(* PLC project ifmCR711S_TemplateProject, CODESYS CODESYS V3.5 SP11 Patch 5 *)
(* stored: creationDateTime 2026-05-10T19:29:40.3172001, version 2.4.10.0, modificationDateTime 2026-05-10T19:24:10.3108894, organization ifm electronic *)
(* Project template with CR711S configured 2.25MByte Standard 2.25MByte Safety *)

(* values of EControlMode: INIT: Initial state when starting ferry *)

{attribute 'qualified_only'}
{attribute 'strict'}
TYPE EControlMode : (INIT, MANUAL, REMOTE, AUTO, REMOTE_MOBILE, FAILSAFE);
END_TYPE

(* values of ETransitionState: STABLE: No switch in progress *)

(* Where the system is in the switch process *)
{attribute 'qualified_only'}
{attribute 'strict'}
TYPE ETransitionState : (INIT, STABLE, PRE_TAKEOVER, VALIDATE_TAKEOVER, FAILSAFE);
END_TYPE

(* values of EPendingMode: NONE: No state pending; PENDING_MANUAL: Pending manual; PENDING_REMOTE: Pending remote; PENDING_AUTO: Pending auto *)

{attribute 'qualified_only'}
{attribute 'strict'}
TYPE EPendingMode : (NONE, PENDING_MANUAL, PENDING_REMOTE, PENDING_AUTO, PENDING_REMOTE_MOBILE);
END_TYPE

PROGRAM PLC_PRG
  VAR
    fbMonitoringChannel : MonitoringChannel;
    fbShutdownService : ShutdownService;
  END_VAR

                    fbMonitoringChannel(
	HB_Manual_OK := EVL.HB_Manual_OK, 
	HB_Remote_OK := EVL.HB_Remote_OK,
	HB_Auto_OK	 := EVL.HB_Auto_OK, 
	HB_Remote_Mobile_OK := EVL.HB_Remote_Mobile_OK
);

fbShutdownService( 
	EmergencyShutdown := fbMonitoringChannel.EmergencyShutdown
); 
                  
END_PROGRAM

FUNCTION_BLOCK MonitoringChannel
  VAR_INPUT
    HB_Manual_OK : BOOL;
    HB_Remote_OK : BOOL;
    HB_Auto_OK : BOOL;
    HB_Remote_Mobile_OK : BOOL;
  END_VAR
  VAR_OUTPUT
    EmergencyShutdown : BOOL;
  END_VAR
  VAR
    HB_Manual_Fail : BOOL;
    HB_Remote_Fail : BOOL;
    HB_Auto_Fail : BOOL;
    HB_Remote_Mobile_Fail : BOOL;
  END_VAR

                    
HB_Manual_Fail := NOT HB_Manual_OK; 
HB_Remote_Fail := NOT HB_Remote_OK; 
HB_Auto_Fail   := NOT HB_Auto_OK;
HB_Remote_Mobile_Fail := NOT HB_Remote_Mobile_OK; 

IF HB_Manual_Fail AND HB_Remote_Fail AND HB_Auto_Fail AND HB_Remote_Mobile_Fail THEN 
	EmergencyShutdown := TRUE; 
END_IF


                  
END_FUNCTION_BLOCK

FUNCTION_BLOCK ShutdownService
  VAR_INPUT
    EmergencyShutdown : BOOL;
  END_VAR
  VAR
    Alert : BOOL;
  END_VAR

                    //Once triggered, the alert stays TRUE until system restart

IF EmergencyShutdown THEN 
	Alert := TRUE; 
END_IF
                  
END_FUNCTION_BLOCK

PROGRAM PLC_PRG
  VAR
    fbInputProcessing : InputProcessing;
    fbControlUnit : ControlUnit;
    fbOutputProcessing : OutputProcessing;
    fbIntegrityCheck : IntegrityCheck;
    fbDecisionLogger : DecisionLogger;
    fbHBGen_Manual : FB_HeartBeatGenerator;
    fbHBGen_Remote : FB_HeartBeatGenerator;
    fbHBGen_Auto : FB_HeartBeatGenerator;
    fbHBGen_Remote_Mobile : FB_HeartBeatGenerator;
    fbHB_Manual : FB_HeartBeat;
    fbHB_Remote : FB_HeartBeat;
    fbHB_Auto : FB_HeartBeat;
    fbHB_Remote_Mobile : FB_HeartBeat;
  END_VAR

                    CR710S_Config(); 			//IO Configuration

IOWrapper.READ_INPUTS(); 	//Call IOWrapper Main Program and Read Data from Inputs   

fbInputProcessing(
	xReqManual 			:= GVL_IO.ReqManual,
	xAckManual 			:= GVL_IO.AckManual, 
	xRelManual 			:= GVL_IO.RelManual, 
	xHB_Manual			:= IN0103.VAR_OUT.xValueDigital, 
	xReqRemote			:= GVL_IO.ReqRemote, 
	xAckRemote			:= GVL_IO.AckRemote, 
	xRelRemote        	:= GVL_IO.RelRemote,
	xHB_Remote        := GVL_HeartBeat.HB_Remote_Signal,
	xReqAuto          := GVL_IO.ReqAuto,
    xAckAuto          := GVL_IO.AckAuto,
    xRelAuto          := GVL_IO.RelAuto,
    xHB_Auto          := GVL_HeartBeat.HB_Auto_Signal,
	xReqRemoteMobile  := GVL_IO.ReqRemoteMobile,
    xAckRemoteMobile  := GVL_IO.AckRemoteMobile,
    xRelRemoteMobile  := GVL_IO.RelRemoteMobile,
    xHB_Remote_Mobile := GVL_HeartBeat.HB_Remote_Mobile_Signal
	
);

fbHB_Manual(xSignal        := fbHBGen_Manual.xSignal);
fbHB_Remote(xSignal        := fbHBGen_Remote.xSignal);
fbHB_Auto(xSignal          := fbHBGen_Auto.xSignal);
fbHB_Remote_Mobile(xSignal := fbHBGen_Remote_Mobile.xSignal);

GVL_HeartBeat.HB_Manual_OK := fbHB_Manual.xOk;
GVL_HeartBeat.HB_Remote_OK := fbHB_Remote.xOk;
GVL_HeartBeat.HB_Auto_OK   := fbHB_Auto.xOk;
GVL_HeartBeat.HB_Remote_Mobile_OK := fbHB_Remote_Mobile.xOk;

//Heartbeat generator
fbHBGen_Manual(); 
fbHBGen_Remote(); 
fbHBGen_Auto();
fbHBGen_Remote_Mobile(); 


fbIntegrityCheck(
    ReqManual        := fbInputProcessing.ReqManual,
    ReqRemote        := fbInputProcessing.ReqRemote,
	ReqAuto			 := fbInputProcessing.ReqAuto,
	ReqRemoteMobile  := fbInputProcessing.ReqRemoteMobile,
    AckManual        := fbInputProcessing.AckManual,
    AckRemote        := fbInputProcessing.AckRemote,
	AckAuto			 := fbInputProcessing.AckAuto,
	AckRemoteMobile  := fbInputProcessing.AckRemoteMobile,
    RelManual        := fbInputProcessing.RelManual,
    RelRemote        := fbInputProcessing.RelRemote,
	RelAuto			 := fbInputProcessing.RelAuto,
	RelRemoteMobile  := fbInputProcessing.RelRemoteMobile,
    HB_Manual_Signal := fbInputProcessing.HB_Manual_Signal,
    HB_Remote_Signal := fbInputProcessing.HB_Remote_Signal,
	HB_Auto_Signal	 := fbInputProcessing.HB_Auto_Signal,
	HB_Remote_Mobile_Signal := fbInputProcessing.HB_Remote_Mobile_Signal, 
);

fbControlUnit(
    ReqManual  		:= fbIntegrityCheck.ReqManual_Out,
	AckManual   	:= fbIntegrityCheck.AckManual_Out,
	RelManual   	:= fbIntegrityCheck.RelManual_Out,
    ReqRemote   	:= fbIntegrityCheck.ReqRemote_Out,
    AckRemote   	:= fbIntegrityCheck.AckRemote_Out,
    RelRemote   	:= fbIntegrityCheck.RelRemote_Out,
	ReqAuto			:= fbIntegrityCheck.ReqAuto_Out,
	AckAuto			:= fbIntegrityCheck.AckAuto_Out,
	RelAuto			:= fbIntegrityCheck.RelAuto_Out,
	ReqRemoteMobile := fbIntegrityCheck.ReqRemoteMobile_Out, 
	AckRemoteMobile := fbIntegrityCheck.AckRemoteMobile_Out, 
	RelRemoteMobile := fbIntegrityCheck.RelRemoteMobile_Out,
	HB_Manual_OK 	:= GVL_HeartBeat.HB_Manual_OK,
	HB_Remote_OK 	:= GVL_HeartBeat.HB_Remote_OK,
	HB_Auto_OK		:= GVL_HeartBeat.HB_Auto_OK, 
	HB_Remote_Mobile_OK := GVL_HeartBeat.HB_Remote_Mobile_OK,
	Valid := fbIntegrityCheck.Valid,
	MaxAckTime := T#10S
);

fbOutputProcessing(
    ReqManual       := fbInputProcessing.ReqManual,
    ReqRemote       := fbInputProcessing.ReqRemote,
	ReqAuto	        := fbInputProcessing.ReqAuto,
	ReqRemoteMobile := fbInputProcessing.ReqRemoteMobile,
    GrantedManual   := fbControlUnit.GrantedManual,
    GrantedRemote   := fbControlUnit.GrantedRemote,
	GrantedAuto	    := fbControlUnit.GrantedAuto,
	GrantedRemoteMobile := fbControlUnit.GrantedRemoteMobile,
	Released 		:= fbControlUnit.Released,
	PendingReady 	:= fbControlUnit.PendingReady,
    Active          := fbControlUnit.Active,
    State           := fbControlUnit.State,
    HB_Manual_OK    := GVL_HeartBeat.HB_Manual_OK,
    HB_Remote_OK    := GVL_HeartBeat.HB_Remote_OK,
	HB_Auto_OK		:= GVL_HeartBeat.HB_Auto_OK,
	HB_Remote_Mobile_OK := GVL_HeartBeat.HB_Remote_Mobile_OK,
);

fbDecisionLogger( 
	Active := fbControlUnit.Active,
	Pending := fbControlUnit.Pending,   
	State := fbControlUnit.State, 
	RejectedRequestFlag := fbControlUnit.RejectedRequestFlag,
	RejectionReason := fbControlUnit.RejectionReason
	
); 
	
OUT0000.VAR_IN.uiValue := SEL(fbOutputProcessing.OUT_GrantedManual, 0, 2500);
OUT0001.VAR_IN.uiValue := SEL(fbOutputProcessing.OUT_GrantedRemote, 0, 2500);
OUT0002.VAR_IN.uiValue := SEL(fbOutputProcessing.OUT_ActiveManual, 0, 2500);
OUT0003.VAR_IN.uiValue := SEL(fbOutputProcessing.OUT_ActiveRemote, 0, 2500);
OUT0004.VAR_IN.uiValue := SEL(fbOutputProcessing.OUT_Pending, 0, 2500);
OUT0005.VAR_IN.uiValue := SEL(fbOutputProcessing.OUT_FailSafe, 0, 2500);
OUT0006.VAR_IN.uiValue := SEL(fbOutputProcessing.OUT_GrantedAuto, 0, 2500);
OUT0007.VAR_IN.uiValue := SEL(fbOutputProcessing.OUT_ActiveAuto, 0, 2500);

GVL_IO.ReleaseRequest_Manual := fbControlUnit.ReleaseRequest_Manual; 
GVL_IO.Releaserequest_Remote := fbControlUnit.ReleaseRequest_Remote; 
GVL_IO.Releaserequest_Auto := fbControlUnit.ReleaseRequest_Auto; 
GVL_IO.ReleaseRequest_Remote_Mobile := fbControlUnit.ReleaseRequest_Remote_Mobile;

EVC.EVL.HB_Manual_OK        := GVL_HeartBeat.HB_Manual_OK;
EVC.EVL.HB_Remote_OK        := GVL_HeartBeat.HB_Remote_OK;
EVC.EVL.HB_Auto_OK          := GVL_HeartBeat.HB_Auto_OK;
EVC.EVL.HB_Remote_Mobile_OK := GVL_HeartBeat.HB_Remote_Mobile_OK;



GVL_State.TimeStamp := GVL_State.TimeStamp + 1; 

IOWrapper.WRITE_OUTPUTS();	//Call IOWrapper Main Program and Write Data to Outputs 
 


                  
END_PROGRAM

PROGRAM CR710S_Config

                    (* IO Configuration*)
config_inputs();
config_outputs();
config_outgroups();


                  

ACTION config_inputs:
                        (* Input Mode Configuration *) // FREQ_SENSE_PERIODS.PERIODS_5, ENCODER_RESOLUTION.EVERY_EDGE
(* Frequency Inputs *)
IN0000.CONFIG.MONITOR		(FILTER_INPUT.UNCHANGED);
IN0001.CONFIG.MONITOR		(FILTER_INPUT.UNCHANGED);
IN0002.CONFIG.MONITOR		(FILTER_INPUT.UNCHANGED);
IN0003.CONFIG.MONITOR		(FILTER_INPUT.UNCHANGED);
IN0500.CONFIG.MONITOR		(FILTER_INPUT.UNCHANGED);
IN0501.CONFIG.MONITOR		(FILTER_INPUT.UNCHANGED);
IN0502.CONFIG.MONITOR		(FILTER_INPUT.UNCHANGED);
IN0503.CONFIG.MONITOR		(FILTER_INPUT.UNCHANGED);

(* Multifuntional Inputs *) 
// MANUAL STATION INPUTS 	
IN0100.CONFIG.IN_DIGITAL_CSI		(FILTER_INPUT.FILTER_5);
IN0101.CONFIG.IN_DIGITAL_CSI		(FILTER_INPUT.FILTER_5);
IN0102.CONFIG.IN_DIGITAL_CSI		(FILTER_INPUT.FILTER_5);
IN0103.CONFIG.IN_DIGITAL_CSI		(FILTER_INPUT.FILTER_1);   
         		
		
IN0600.CONFIG.MONITOR		(FILTER_INPUT.FILTER_5);
IN0601.CONFIG.MONITOR		(FILTER_INPUT.FILTER_5);
IN0602.CONFIG.MONITOR		(FILTER_INPUT.FILTER_5);
IN0603.CONFIG.MONITOR		(FILTER_INPUT.FILTER_1);

(* Resistopr Inputs *)      	
IN0400.CONFIG.MONITOR		(FILTER_INPUT.UNCHANGED);
IN0401.CONFIG.MONITOR		(FILTER_INPUT.UNCHANGED);
IN0900.CONFIG.MONITOR		(FILTER_INPUT.UNCHANGED);
IN0901.CONFIG.MONITOR		(FILTER_INPUT.UNCHANGED);

(* Diagnostic and Protection Configuration *) //eDIAG_PROT_MODE.DIAG_PROT
(* Frequency Inputs *) 
IN0000.CONFIG.SET_DIAG_LVL_PROT		(0, 32000, 100, eDIAG_PROT_MODE.DIAG_PROT);
IN0001.CONFIG.SET_DIAG_LVL_PROT		(0, 32000, 100, eDIAG_PROT_MODE.DIAG_PROT);
IN0002.CONFIG.SET_DIAG_LVL_PROT		(0, 32000, 100, eDIAG_PROT_MODE.DIAG_PROT);
IN0003.CONFIG.SET_DIAG_LVL_PROT		(0, 32000, 100, eDIAG_PROT_MODE.DIAG_PROT);
IN0500.CONFIG.SET_DIAG_LVL_PROT		(0, 32000, 100, eDIAG_PROT_MODE.DIAG_PROT);
IN0501.CONFIG.SET_DIAG_LVL_PROT		(0, 32000, 100, eDIAG_PROT_MODE.DIAG_PROT);
IN0502.CONFIG.SET_DIAG_LVL_PROT		(0, 32000, 100, eDIAG_PROT_MODE.DIAG_PROT);
IN0503.CONFIG.SET_DIAG_LVL_PROT		(0, 32000, 100, eDIAG_PROT_MODE.DIAG_PROT);
(* Multifuntional Inputs *)                          
IN0100.CONFIG.SET_DIAG_LVL_PROT		(0, 32000, 100, eDIAG_PROT_MODE.DIAG_PROT);
IN0101.CONFIG.SET_DIAG_LVL_PROT		(0, 32000, 100, eDIAG_PROT_MODE.DIAG_PROT);
IN0102.CONFIG.SET_DIAG_LVL_PROT		(0, 32000, 100, eDIAG_PROT_MODE.DIAG_PROT);
IN0103.CONFIG.SET_DIAG_LVL_PROT		(0, 32000, 100, eDIAG_PROT_MODE.DIAG_PROT);                                                    
IN0600.CONFIG.SET_DIAG_LVL_PROT		(0, 32000, 100, eDIAG_PROT_MODE.DIAG_PROT);
IN0601.CONFIG.SET_DIAG_LVL_PROT		(0, 32000, 100, eDIAG_PROT_MODE.DIAG_PROT);
IN0602.CONFIG.SET_DIAG_LVL_PROT		(0, 32000, 100, eDIAG_PROT_MODE.DIAG_PROT);
IN0603.CONFIG.SET_DIAG_LVL_PROT		(0, 32000, 100, eDIAG_PROT_MODE.DIAG_PROT);
(* Resistopr Inputs *)                               
IN0400.CONFIG.SET_DIAG_LVL_PROT		(0, 32000, 100, eDIAG_PROT_MODE.DIAG_PROT);
IN0401.CONFIG.SET_DIAG_LVL_PROT		(0, 32000, 100, eDIAG_PROT_MODE.DIAG_PROT);
IN0900.CONFIG.SET_DIAG_LVL_PROT		(0, 32000, 100, eDIAG_PROT_MODE.DIAG_PROT);
IN0901.CONFIG.SET_DIAG_LVL_PROT		(0, 32000, 100, eDIAG_PROT_MODE.DIAG_PROT);

(* Digital Switching Threshold - Default ON:= 0.7*Vbb, OFF:= 0.3*Vbb *)
(* Frequency Inputs *) 
IN0000.CONFIG.SET_SWITCH_THRESHOLD(300, 700); // 300 = 30% - 700 = 70%
IN0001.CONFIG.SET_SWITCH_THRESHOLD(300, 700);
IN0002.CONFIG.SET_SWITCH_THRESHOLD(300, 700);
IN0003.CONFIG.SET_SWITCH_THRESHOLD(300, 700);
IN0500.CONFIG.SET_SWITCH_THRESHOLD(300, 700);
IN0501.CONFIG.SET_SWITCH_THRESHOLD(300, 700);
IN0502.CONFIG.SET_SWITCH_THRESHOLD(300, 700);
IN0503.CONFIG.SET_SWITCH_THRESHOLD(300, 700);
(* Multifuntional Inputs *)   
IN0100.CONFIG.SET_SWITCH_THRESHOLD(300, 700);
IN0101.CONFIG.SET_SWITCH_THRESHOLD(300, 700);
IN0102.CONFIG.SET_SWITCH_THRESHOLD(300, 700);
IN0103.CONFIG.SET_SWITCH_THRESHOLD(300, 700);
IN0600.CONFIG.SET_SWITCH_THRESHOLD(300, 700);
IN0601.CONFIG.SET_SWITCH_THRESHOLD(300, 700);
IN0602.CONFIG.SET_SWITCH_THRESHOLD(300, 700);
IN0603.CONFIG.SET_SWITCH_THRESHOLD(300, 700);
(* Resistopr Inputs *)     
IN0400.CONFIG.SET_SWITCH_THRESHOLD(300, 700);
IN0401.CONFIG.SET_SWITCH_THRESHOLD(300, 700);
IN0900.CONFIG.SET_SWITCH_THRESHOLD(300, 700);
IN0901.CONFIG.SET_SWITCH_THRESHOLD(300, 700);
                      
END_ACTION

ACTION config_outgroups:
                        (* Output Group Mode Configuration *) 
OUTGROUP0.CONFIG.MONITOR				(FILTER_OUTPUT_GROUP.UNCHANGED);
OUTGROUP1.CONFIG.MONITOR				(FILTER_OUTPUT_GROUP.UNCHANGED);

(* Diagnostic and Protection Configuration *) 
OUTGROUP0.CONFIG.SET_DIAG_LVL_PROT		(0, 12000, 100, eDIAG_PROT_MODE.DIAG_PROT);
OUTGROUP1.CONFIG.SET_DIAG_LVL_PROT		(0, 12000, 100, eDIAG_PROT_MODE.DIAG_PROT);

                      
END_ACTION

ACTION config_outputs:
                        (* Output Mode Configuration *) 
(* Group 0 *) //ÄNDRAT HÄR?? Osäker om dessa stämmer? 
OUT0000.CONFIG.OUT_DIGITAL_CSO				(FILTER_OUTPUT.UNCHANGED);
OUT0001.CONFIG.OUT_DIGITAL_CSO				(FILTER_OUTPUT.UNCHANGED);
OUT0002.CONFIG.OUT_DIGITAL_CSO				(FILTER_OUTPUT.UNCHANGED);
OUT0003.CONFIG.OUT_DIGITAL_CSO				(FILTER_OUTPUT.UNCHANGED);
OUT0004.CONFIG.OUT_DIGITAL_CSO				(FILTER_OUTPUT.UNCHANGED);
OUT0005.CONFIG.OUT_DIGITAL_CSO				(FILTER_OUTPUT.UNCHANGED);
OUT0006.CONFIG.OUT_DIGITAL_CSO				(FILTER_OUTPUT.UNCHANGED);
OUT0007.CONFIG.OUT_DIGITAL_CSO				(FILTER_OUTPUT.UNCHANGED);

(* Group 1 *)         				    		
OUT0100.CONFIG.MONITOR			(FILTER_OUTPUT.UNCHANGED);
OUT0101.CONFIG.MONITOR			(FILTER_OUTPUT.UNCHANGED);
OUT0102.CONFIG.MONITOR			(FILTER_OUTPUT.UNCHANGED);
OUT0103.CONFIG.MONITOR			(FILTER_OUTPUT.UNCHANGED);
OUT0104.CONFIG.MONITOR			(FILTER_OUTPUT.UNCHANGED);
OUT0105.CONFIG.MONITOR			(FILTER_OUTPUT.UNCHANGED);
OUT0106.CONFIG.MONITOR			(FILTER_OUTPUT.UNCHANGED);
OUT0107.CONFIG.MONITOR			(FILTER_OUTPUT.UNCHANGED);

(* Output SensorSupply and Analogue *)      				
OUT3000.CONFIG.MONITOR			(FILTER_OUTPUT.UNCHANGED);
OUT3001.CONFIG.MONITOR			(FILTER_OUTPUT.UNCHANGED);	

(* Diagnostic and Protection Configuration *) 
(* Group 0 *)
OUT0000.CONFIG.SET_DIAG_LVL_PROT	(0, 2500, 100, eDIAG_PROT_MODE.DIAG_PROT);
OUT0001.CONFIG.SET_DIAG_LVL_PROT	(0, 2500, 100, eDIAG_PROT_MODE.DIAG_PROT);
OUT0002.CONFIG.SET_DIAG_LVL_PROT	(0, 2500, 100, eDIAG_PROT_MODE.DIAG_PROT);
OUT0003.CONFIG.SET_DIAG_LVL_PROT	(0, 2500, 100, eDIAG_PROT_MODE.DIAG_PROT);
OUT0004.CONFIG.SET_DIAG_LVL_PROT	(0, 2500, 100, eDIAG_PROT_MODE.DIAG_PROT);
OUT0005.CONFIG.SET_DIAG_LVL_PROT	(0, 2500, 100, eDIAG_PROT_MODE.DIAG_PROT);
OUT0006.CONFIG.SET_DIAG_LVL_PROT	(0, 4000, 100, eDIAG_PROT_MODE.DIAG_PROT);
OUT0007.CONFIG.SET_DIAG_LVL_PROT	(0, 4000, 100, eDIAG_PROT_MODE.DIAG_PROT);
(* Group 1 *)                                       
OUT0100.CONFIG.SET_DIAG_LVL_PROT	(0, 2500, 100, eDIAG_PROT_MODE.DIAG_PROT);
OUT0101.CONFIG.SET_DIAG_LVL_PROT	(0, 2500, 100, eDIAG_PROT_MODE.DIAG_PROT);
OUT0102.CONFIG.SET_DIAG_LVL_PROT	(0, 2500, 100, eDIAG_PROT_MODE.DIAG_PROT);
OUT0103.CONFIG.SET_DIAG_LVL_PROT	(0, 2500, 100, eDIAG_PROT_MODE.DIAG_PROT);
OUT0104.CONFIG.SET_DIAG_LVL_PROT	(0, 2500, 100, eDIAG_PROT_MODE.DIAG_PROT);
OUT0105.CONFIG.SET_DIAG_LVL_PROT	(0, 2500, 100, eDIAG_PROT_MODE.DIAG_PROT);
OUT0106.CONFIG.SET_DIAG_LVL_PROT	(0, 4000, 100, eDIAG_PROT_MODE.DIAG_PROT);
OUT0107.CONFIG.SET_DIAG_LVL_PROT	(0, 4000, 100, eDIAG_PROT_MODE.DIAG_PROT);

                      
END_ACTION
END_PROGRAM

FUNCTION_BLOCK FB_HeartBeat
  VAR_INPUT
    xSignal : BOOL;
  END_VAR
  VAR_OUTPUT
    xOk : BOOL;
  END_VAR
  VAR
    tonTimeout : TON;
    xPrevSignal : BOOL;
    xPulse : BOOL;
  END_VAR

                    xPulse := (xSignal <> xPrevSignal);
xPrevSignal := xSignal;
// Om ingen ny puls kommer, låt timern gå 
tonTimeout(IN := NOT xPulse, PT := GVL_HeartBeat.HB_Monitor_Timeout);
xOk := NOT tonTimeout.Q;

                  
END_FUNCTION_BLOCK

FUNCTION_BLOCK ControlUnit
  VAR_INPUT
    Valid : BOOL;
    ReqManual : BOOL;
    ReqRemote : BOOL;
    ReqAuto : BOOL;
    ReqRemoteMobile : BOOL;
    AckManual : BOOL;
    AckRemote : BOOL;
    AckAuto : BOOL;
    AckRemoteMobile : BOOL;
    RelManual : BOOL;
    RelRemote : BOOL;
    RelAuto : BOOL;
    RelRemoteMobile : BOOL;
    HB_Manual_OK : BOOL;
    HB_Remote_OK : BOOL;
    HB_Auto_OK : BOOL;
    HB_Remote_Mobile_OK : BOOL;
    Velocity : REAL;  (* Still needed? *)
    MaxVelocity : REAL;
    SteeringAngle : REAL;
    MaxSteering : REAL;
    MaxAckTime : TIME;  (* timeout threshold *)
  END_VAR
  VAR_OUTPUT
    Active : EControlMode := EControlMode.INIT;  (* Ändrade från manual->init *)
    GrantedManual : BOOL;
    GrantedRemote : BOOL;
    GrantedAuto : BOOL;
    GrantedRemoteMobile : BOOL;
    State : ETransitionState;
    Released : BOOL;
    PendingReady : BOOL;
    RejectedRequestFlag : BOOL;
    RejectionReason : STRING;
    ReleaseRequest_Manual : BOOL;
    ReleaseRequest_Remote : BOOL;
    ReleaseRequest_Auto : BOOL;
    ReleaseRequest_Remote_Mobile : BOOL;
  END_VAR
  VAR
    Pending : EPendingMode;
    tAckTimer : TON;
    xReqRemoteOld : BOOL := FALSE;
    xReqManualOld : BOOL := FALSE;
    xReqAutoOld : BOOL := FALSE;
    xReqRemoteMobileOld : BOOL := FALSE;
    xReqRemotePulse : BOOL := FALSE;
    xReqManualPulse : BOOL := FALSE;
    xReqAutoPulse : BOOL := FALSE;
    xReqRemoteMobilePulse : BOOL := FALSE;
    xPendingManualLatch : BOOL := FALSE;
    xPendingRemoteLatch : BOOL := FALSE;
    xPendingAutoLatch : BOOL := FALSE;
    xPendingRemoteMobileLatch : BOOL := FALSE;
  END_VAR

                    //Detect when a request signal goes from FALSE to TRUE
//Ensures each request is only processed once per button press
xReqRemotePulse := ReqRemote AND NOT xReqRemoteOld; 
xReqManualPulse := ReqManual AND NOT xReqManualOld; 
xReqAutoPulse := ReqAuto AND NOT xReqAutoOld; 
xReqRemoteMobilePulse := ReqRemoteMobile AND NOT xReqRemoteMobileOld; 

//Store previous signal state for next scan's edge detection
xReqRemoteOld := ReqRemote; 
xReqManualOld := ReqManual; 
xReqAutoOld := ReqAuto; 
xReqRemoteMobileOld := ReqRemoteMobile; 

//Safety guard - if active loses heartbeat force FAILSAFE immediately
//This check runs every scan before the state machine, acting as an interrupt
IF (Active = EControlMode.REMOTE AND NOT HB_Remote_OK) OR 
	(Active = EControlMode.MANUAL AND NOT HB_Manual_OK) OR 
	(Active = EControlMode.AUTO AND NOT HB_Auto_OK) OR 
	(Active = EControlMode.REMOTE_MOBILE AND NOT HB_Remote_Mobile_OK) THEN
	Active 	:= EControlMode.FAILSAFE; 
	Pending := EPendingMode.NONE; 
	State 	:= ETransitionState.FAILSAFE; 
	GrantedManual 		:= FALSE;
	GrantedRemote 		:= FALSE;
	GrantedAuto 		:= FALSE;
	GrantedRemoteMobile := FALSE; 
	RETURN; 
END_IF 

//Safety guard - if IntegrityCheck detected invalid signal combination force FAILSAFE
//Prevents corrupted or contradictiory signals from reaching decision logic
IF NOT Valid THEN
	Active 			:=  EControlMode.FAILSAFE;
	Pending 		:= EPendingMode.NONE;
	State 			:= ETransitionState.FAILSAFE;
	PendingReady 	:= FALSE;
	Released 		:= FALSE;
	tAckTimer(IN := FALSE, PT := MaxAckTime);
	GrantedManual := FALSE;
	GrantedRemote := FALSE;
	GrantedAuto := FALSE;
	GrantedRemoteMobile := FALSE; 
	RejectedRequestFlag := TRUE;
	RejectionReason := 'FAILSAFE: INVALID_SIGNAL';
	RETURN;	
END_IF

//Main state machine - contrls transitions between control stations
//States: INIT -> STABLE <-> PRE_TAKEOVER <-> VALIDATE_TAKEOVER, any state -> FAILSAFE
CASE State OF
	//INIT - system startup, waiting for the first valid request
	//System remains here until a station with valid heartbeat requests control 
	ETransitionState.INIT:
		IF xReqManualPulse AND HB_Manual_OK THEN
            Active := EControlMode.MANUAL;
            State  := ETransitionState.STABLE;
        ELSIF xReqRemotePulse AND HB_Remote_OK THEN
            Active := EControlMode.REMOTE;
            State  := ETransitionState.STABLE;
        ELSIF xReqAutoPulse AND HB_Auto_OK THEN
            Active := EControlMode.AUTO;
            State  := ETransitionState.STABLE;
		ELSIF xReqRemoteMobilePulse AND HB_Remote_Mobile_OK THEN 
			Active := EControlMode.REMOTE_MOBILE; 
			State := ETransitionState.STABLE; 
        END_IF 
	
	// FAILSAFE - terminal error state, no transitions allowed
	// Entered when heartbeat is lost, signals are invalid or internal inconsistency detected
	//Requires manual intervention to recover	
	ETransitionState.FAILSAFE:
		Pending       	:= EPendingMode.NONE;
		PendingReady	:= FALSE;
		Released 		:= FALSE;
		tAckTimer(IN := FALSE, PT := MaxAckTime);
	
	//STABLE - normal operating state, one station is active, no transition in progress
	// Resets rejection flags and waits for a new takeover request	
	ETransitionState.STABLE: 
		Pending := EPendingMode.NONE; 
		tAckTimer(IN := FALSE, PT := MaxAckTime);
		RejectedRequestFlag := FALSE; 
		RejectionReason := ''; 
		
		//Priority order dor simultaneius requests: MANUAL > REMOTE > AUTO > REMOTE_MOBILE
		//Documented in ADR-X - simultaneous requests from different stations
		IF xReqManualPulse THEN 
			xPendingManualLatch := TRUE; 
			State := ETransitionState.PRE_TAKEOVER; 
		ELSIF xReqRemotePulse THEN 
			xPendingRemoteLatch := TRUE; 
			State := ETransitionState.PRE_TAKEOVER; 
		ELSIF xReqAutoPulse THEN 
			xPendingAutoLatch := TRUE; 
			State := ETransitionState.PRE_TAKEOVER; 
		ELSIF xReqRemoteMobilePulse THEN 
			xPendingRemoteMobileLatch := TRUE; 
			State := ETransitionState.PRE_TAKEOVER; 
		END_IF
	
	//PRE_TAKEOVER - validates wheter a takover request can proceed
	//Checks that requesting station is not already active and has valid heartbeat
	//Rejected request are logged with reason
	ETransitionState.PRE_TAKEOVER:	
		IF xPendingManualLatch AND Active <> EControlMode.MANUAL AND HB_Manual_OK THEN 
			Pending := EPendingMode.PENDING_MANUAL; 
			State 	:= ETransitionState.VALIDATE_TAKEOVER; 
		ELSIF xPendingRemoteLatch AND Active <> EControlMode.REMOTE AND HB_Remote_OK THEN 
			Pending := EPendingMode.PENDING_REMOTE; 
			State 	:= ETransitionState.VALIDATE_TAKEOVER; 
		ELSIF xPendingAutoLatch AND Active <> EControlMode.AUTO AND HB_Auto_OK THEN 
			Pending := EPendingMode.PENDING_AUTO; 
			State 	:= ETransitionState.VALIDATE_TAKEOVER; 
		ELSIF xPendingRemoteMobileLatch AND Active <> EControlMode.REMOTE_MOBILE AND HB_Remote_Mobile_OK THEN 
			Pending := EPendingMode.PENDING_REMOTE_MOBILE; 
			State	:= ETransitionState.VALIDATE_TAKEOVER; 
		ELSE 
			//Request rejected - log reason for decision logger
			Pending := EPendingMode.NONE; 
			State := ETransitionState.STABLE; 
			RejectedRequestFlag := TRUE; 
			IF (xPendingManualLatch AND NOT HB_Manual_OK) OR 
				(xPendingRemoteLatch AND NOT HB_Remote_OK) OR 
				(xPendingAutoLatch AND NOT HB_Auto_OK) OR 
				(xPendingRemoteMobileLatch AND NOT HB_Remote_Mobile_OK) THEN 
					RejectionReason := 'Request rejected: Heartbeat failure'; 
			ELSIF (xPendingManualLatch AND Active = EControlMode.MANUAL) OR 
				(xPendingRemoteLatch AND Active = EControlMode.REMOTE) OR
				(xPendingAutoLatch AND Active = EControlMode.AUTO) OR 
				(xPendingRemoteMobileLatch AND Active = EControlMode.REMOTE_MOBILE) THEN  
					RejectionReason := 'Request rejection: Station already active'; 
			ELSE 
					RejectionReason := 'Request rejected: Conflicting request'; 
			END_IF
		END_IF
		
		//Clear all latches regardless of outcome - each request is only evaluated once
		xPendingManualLatch := FALSE; 
		xPendingRemoteLatch := FALSE; 
		xPendingAutoLatch 	:= FALSE;
		xPendingRemoteMobileLatch := FALSE; 
		
	
	//VALIDATE_TAKEOVER - handshake phase, waiting for release from active and ack from pending
	//Transition completes when active station releases and pending station acknowledges
	//Aborted if heartbeat is lost or acknowledgement timer expires
	ETransitionState.VALIDATE_TAKEOVER: 
		
		ReleaseRequest_Manual := (Active = EControlMode.MANUAL); 
		ReleaseRequest_Remote := (Active = EControlMode.REMOTE); 
		ReleaseRequest_Auto := (Active = EControlMode.AUTO); 
		ReleaseRequest_Remote_Mobile := (Active = EControlMode.REMOTE_MOBILE);
		
		tAckTimer(IN := TRUE, PT := MaxAckTime); 
		
		//Stop transition if the new station loses connection or cancels its request
		IF (Pending = EPendingMode.PENDING_MANUAL AND (NOT ReqManual OR NOT HB_Manual_OK)) OR
			(Pending = EPendingMode.PENDING_REMOTE AND (NOT ReqRemote OR NOT HB_Remote_OK)) OR 
			(Pending = EPendingMode.PENDING_AUTO AND (NOT ReqAuto OR NOT HB_Auto_OK)) OR 
			(Pending = EPendingMode.PENDING_REMOTE_MOBILE AND (NOT ReqRemoteMobile OR NOT HB_Remote_Mobile_OK)) THEN  
			Pending := EPendingMode.NONE; 
			State := ETransitionState.STABLE; 
			tAckTimer (IN := FALSE, PT := MaxAckTime); // Reset timer
			PendingReady := FALSE;
			Released := FALSE;
			ReleaseRequest_Manual := FALSE; 
			ReleaseRequest_Remote := FALSE; 
			ReleaseRequest_Auto := FALSE; 
			ReleaseRequest_Remote_Mobile := FALSE; 
			RejectedRequestFlag := TRUE; 
			RejectionReason := 'Request rejected: Heartbeat loss during handover'; 
		
		//Abort - pending station did not acknowledge within allowed time
		ELSIF tAckTimer.Q THEN 
			Pending := EPendingMode.NONE; 
			State := ETransitionState.STABLE; 
			tAckTimer(IN := FALSE, PT := MaxAckTime); 
			PendingReady := FALSE;
			Released := FALSE;
			ReleaseRequest_Manual := FALSE; 
			ReleaseRequest_Remote := FALSE; 
			ReleaseRequest_Auto := FALSE; 
			ReleaseRequest_Remote_Mobile := FALSE; 
			RejectedRequestFlag := TRUE; 
			RejectionReason := 'Request rejected: acknowledgement timeout'; 
			
		ELSE
			//Read release signal from active station
			Released := FALSE;
			CASE Active OF 
				EControlMode.MANUAL: Released := RelManual; 
				EControlMode.REMOTE: Released := RelRemote; 
				EControlMode.AUTO: Released := RelAuto; 
				EControlMode.REMOTE_MOBILE: Released := RelRemoteMobile; 
			END_CASE	
			
			//Read acknowledgement from pending station
			PendingReady := FALSE;
			CASE Pending OF 
				EPendingMode.PENDING_MANUAL: PendingReady := AckManual; 
				EPendingMode.PENDING_REMOTE: PendingReady := AckRemote; 
				EPendingMode.PENDING_AUTO: PendingReady := AckAuto; 
				EPendingMode.PENDING_REMOTE_MOBILE: PendingReady := AckRemoteMobile; 
			END_CASE

			//Safety check: the new station must not be the same as the current one
			//PRE_TAKEOVER prevents this, but if reached here it indicates internal fault
			IF (Pending = EPendingMode.PENDING_MANUAL AND Active = EControlMode.MANUAL) OR
				(Pending = EPendingMode.PENDING_REMOTE AND Active = EControlMode.REMOTE) OR
				(Pending = EPendingMode.PENDING_AUTO AND Active = EControlMode.AUTO) OR
				(Pending = EPendingMode.PENDING_REMOTE_MOBILE AND Active = EControlMode.REMOTE_MOBILE) THEN
					Active 			:= EControlMode.FAILSAFE;
					Pending 		:= EPendingMode.NONE;
					State			:= ETransitionState.FAILSAFE;
					PendingReady 	:= FALSE;
					Released		:= FALSE;
					tAckTimer(IN := FALSE, PT := MaxAckTime);
					GrantedManual 	:= FALSE;
					GrantedRemote 	:= FALSE;
					GrantedAuto 	:= FALSE;
					GrantedRemoteMobile := FALSE;
					ReleaseRequest_Manual := FALSE; 
					ReleaseRequest_Remote := FALSE; 
					ReleaseRequest_Auto := FALSE; 
					ReleaseRequest_Remote_Mobile := FALSE;  
					RejectedRequestFlag := TRUE; 
					RejectionReason := 'Request rejected: Integrity violation, pending matches active';
					RETURN;		
			END_IF
			
			//Complete transition - both conditions met
			IF Released AND PendingReady THEN 
				CASE Pending OF
					EPendingMode.PENDING_MANUAL: Active := EControlMode.MANUAL; 
					EPendingMode.PENDING_REMOTE: Active := EControlMode.REMOTE; 
					EPendingMode.PENDING_AUTO: Active := EControlMode.AUTO; 
					EPendingMode.PENDING_REMOTE_MOBILE: Active := EControlMode.REMOTE_MOBILE; 
				END_CASE
				Pending := EPendingMode.NONE; 
				State := ETransitionState.STABLE; 
				tAckTimer(IN := FALSE, PT := MaxAckTime); 
				PendingReady := FALSE;
				Released := FALSE; 
				ReleaseRequest_Manual := FALSE; 
				ReleaseRequest_Remote := FALSE; 
				ReleaseRequest_Auto := FALSE; 
				ReleaseRequest_Remote_Mobile := FALSE; 
			END_IF
	END_IF
END_CASE

//Grant signals - updated each scan based on current pending mode
//Stations use these to know their request has been approved
GrantedManual := (Pending = EPendingMode.PENDING_MANUAL);
GrantedRemote := (Pending = EPendingMode.PENDING_REMOTE);
GrantedAuto   := (Pending = EPendingMode.PENDING_AUTO);
GrantedRemoteMobile := (Pending = EPendingMode.PENDING_REMOTE_MOBILE); 


                  
END_FUNCTION_BLOCK

FUNCTION_BLOCK InputProcessing
  VAR_INPUT
    xReqRemote : BOOL;
    xAckRemote : BOOL;
    xRelRemote : BOOL;
    xHB_Remote : BOOL;
    xReqManual : BOOL;
    xAckManual : BOOL;
    xRelManual : BOOL;
    xHB_Manual : BOOL;
    xReqAuto : BOOL;
    xAckAuto : BOOL;
    xRelAuto : BOOL;
    xHB_Auto : BOOL;
    xReqRemoteMobile : BOOL;
    xAckRemoteMobile : BOOL;
    xRelRemoteMobile : BOOL;
    xHB_Remote_Mobile : BOOL;
  END_VAR
  VAR_OUTPUT
    ReqManual : BOOL;
    AckManual : BOOL;
    RelManual : BOOL;
    HB_Manual_Signal : BOOL;
    ReqRemote : BOOL;
    AckRemote : BOOL;
    RelRemote : BOOL;
    HB_Remote_Signal : BOOL;
    ReqAuto : BOOL;
    AckAuto : BOOL;
    RelAuto : BOOL;
    HB_Auto_Signal : BOOL;
    ReqRemoteMobile : BOOL;
    AckRemoteMobile : BOOL;
    RelRemoteMobile : BOOL;
    HB_Remote_Mobile_Signal : BOOL;
  END_VAR

                    // Manual input - with an added abstraction layer after the hardware channels
ReqManual := xReqManual; 
AckManual := xAckManual; 
RelManual := xRelManual; 
HB_Manual_Signal := xHB_Manual; 

// Remote input - from BOOL input
ReqRemote := xReqRemote; 
AckRemote := xAckRemote; 
RelRemote := xRelRemote; 
HB_Remote_Signal := xHB_Remote;

// Autonomous input - from BOOL input
ReqAuto	 := xReqAuto;
AckAuto	 := xAckAuto;
RelAuto	 := xRelAuto;
HB_Auto_Signal   := xHB_Auto;

// Remote mobile - from BOOL input
ReqRemoteMobile := xReqRemoteMobile; 
AckRemoteMobile := xAckRemoteMobile; 
RelRemoteMobile := xRelRemoteMobile;
HB_Remote_Mobile_Signal := xHB_Remote_Mobile; 

                  
END_FUNCTION_BLOCK

FUNCTION_BLOCK OutputProcessing
  VAR_INPUT
    ReqManual : BOOL;
    ReqRemote : BOOL;
    ReqAuto : BOOL;
    ReqRemoteMobile : BOOL;
    GrantedManual : BOOL;
    GrantedRemote : BOOL;
    GrantedAuto : BOOL;
    GrantedRemoteMobile : BOOL;
    Released : BOOL;
    PendingReady : BOOL;
    Active : EControlMode;
    State : ETransitionState;
    HB_Manual_OK : BOOL;
    HB_Remote_OK : BOOL;
    HB_Auto_OK : BOOL;
    HB_Remote_Mobile_OK : BOOL;
    RejectedRequestFlag : BOOL;
  END_VAR
  VAR_OUTPUT
    OUT_GrantedManual : BOOL;
    OUT_GrantedRemote : BOOL;
    OUT_GrantedAuto : BOOL;
    OUT_GrantedRemoteMobile : BOOL;
    OUT_ActiveManual : BOOL;
    OUT_ActiveRemote : BOOL;
    OUT_ActiveAuto : BOOL;
    OUT_ActiveRemoteMobile : BOOL;
    OUT_Pending : BOOL;
    OUT_PendingReady : BOOL;
    OUT_Released : BOOL;
    OUT_NoHB_Manual : BOOL;  (* loss of heartbeat *)
    OUT_NoHB_Remote : BOOL;  (* loss of heartbeat *)
    OUT_NoHB_Auto : BOOL;  (* loss of heartbeat *)
    OUT_NoHB_RemoteMobile : BOOL;
    OUT_FailSafe : BOOL;
    OUT_State_Stable : BOOL;
    OUT_State_Validate : BOOL;
    OUT_State_FailSafe : BOOL;
    OUT_RejectedRequestFlag : BOOL;
  END_VAR

                    //No outputs are active during INIT or FAILSAFE
IF Active = EControlMode.INIT OR Active = EControlMode.FAILSAFE THEN 
	OUT_ActiveManual := FALSE; 
	OUT_ActiveRemote  := FALSE;
	OUT_ActiveAuto    := FALSE;
	OUT_ActiveRemoteMobile := FALSE; 
	OUT_GrantedManual := FALSE; 
	OUT_GrantedRemote := FALSE; 
	OUT_GrantedAuto	  := FALSE;
	OUT_GrantedRemoteMobile := FALSE; 
	OUT_Pending		  := FALSE; 
	OUT_PendingReady  := FALSE; 
	OUT_Released	  := FALSE; 
ELSE
	OUT_GrantedManual := GrantedManual; 
	OUT_GrantedRemote := GrantedRemote; 
	OUT_GrantedAuto	  := GrantedAuto;
	OUT_GrantedRemoteMobile := GrantedRemoteMobile; 
	OUT_ActiveManual  := (Active = EControlMode.MANUAL); 
	OUT_ActiveRemote  := (Active = EControlMode.REMOTE);
	OUT_ActiveAuto    := (Active = EControlMode.AUTO);
	OUT_ActiveRemoteMobile := (Active = EControlMode.REMOTE_MOBILE); 
	OUT_Pending		  := (State = ETransitionState.VALIDATE_TAKEOVER) OR 
						 (State = ETransitionState.PRE_TAKEOVER); 
	OUT_PendingReady  := PendingReady; 
	OUT_Released	  := Released; 
END_IF
OUT_FailSafe	  := (Active = EControlMode.FAILSAFE);  
OUT_RejectedRequestFlag := RejectedRequestFlag; 
//Heartbeat should be visible regardless of mode we're in
OUT_NoHB_Manual   := NOT HB_Manual_OK; 
OUT_NoHB_Remote   := NOT HB_Remote_OK; 
OUT_NoHB_Auto	  := NOT HB_Auto_OK;
OUT_NoHB_RemoteMobile := NOT HB_Remote_Mobile_OK; 

OUT_State_Stable := (State = ETransitionState.STABLE); 
OUT_State_Validate := (State = ETransitionState.VALIDATE_TAKEOVER); 
OUT_State_FailSafe := (State = ETransitionState.FAILSAFE); 


                  
END_FUNCTION_BLOCK

FUNCTION_BLOCK FB_HeartBeatGenerator
  VAR_OUTPUT
    xSignal : BOOL;
  END_VAR
  VAR
    tonToggle : TON;
    xEnable : BOOL := TRUE;
  END_VAR

                    //Start timer
tonToggle(IN := xEnable, PT := T#200MS);

//När timer gått, växla signal
IF tonToggle.Q THEN
	xSignal 		:= NOT xSignal;
	tonToggle(IN 	:= FALSE, PT := GVL_HeartBeat.HB_Generator_Interval);
	xEnable 		:= TRUE;
END_IF;

//Heartbeat-generatorns intervall och heartbeat-monitorns 
//timeout är två separata värden utan formell koppling.
// Om något värde ändras utan att det andra justeras kan
// heartbeat-detektionen sluta fungera.
                  
END_FUNCTION_BLOCK

FUNCTION_BLOCK IntegrityCheck
  VAR_INPUT
    ReqManual : BOOL;
    ReqRemote : BOOL;
    ReqAuto : BOOL;
    ReqRemoteMobile : BOOL;
    AckManual : BOOL;
    AckRemote : BOOL;
    AckAuto : BOOL;
    AckRemoteMobile : BOOL;
    RelManual : BOOL;
    RelRemote : BOOL;
    RelAuto : BOOL;
    RelRemoteMobile : BOOL;
    HB_Manual_Signal : BOOL;
    HB_Remote_Signal : BOOL;
    HB_Auto_Signal : BOOL;
    HB_Remote_Mobile_Signal : BOOL;
  END_VAR
  VAR_OUTPUT
    Valid : BOOL;  (* All signals passed sanity check *)
    ReqManual_Out : BOOL;
    ReqRemote_Out : BOOL;
    ReqAuto_Out : BOOL;
    ReqRemoteMobile_Out : BOOL;
    AckManual_Out : BOOL;
    AckRemote_Out : BOOL;
    AckAuto_Out : BOOL;
    AckRemoteMobile_Out : BOOL;
    RelManual_Out : BOOL;
    RelRemote_Out : BOOL;
    RelAuto_Out : BOOL;
    RelRemoteMobile_Out : BOOL;
    HB_Manual_Out : BOOL;
    HB_Remote_Out : BOOL;
    HB_Auto_Out : BOOL;
    HB_Remote_Mobile_Out : BOOL;
  END_VAR

                    IF (ReqManual AND RelManual) OR //a station requesting and releasing at the same time
   (ReqRemote AND RelRemote) OR
   (ReqAuto AND RelAuto) OR
   (ReqRemoteMobile AND RelRemoteMobile) OR 
   (AckManual AND RelManual) OR //Station acknowledging and releasing simutaneously 
   (AckRemote AND RelRemote) OR
   (AckAuto AND RelAuto) OR
   (AckRemoteMobile AND RelRemoteMobile) THEN
   	Valid        := FALSE; 
    ReqManual_Out := FALSE;
    ReqRemote_Out := FALSE;
	ReqAuto_Out	  := FALSE;
	ReqRemoteMobile_Out := FALSE; 
    AckManual_Out := FALSE;
    AckRemote_Out := FALSE;
	AckAuto_Out	  := FALSE;
	AckRemoteMobile_Out := FALSE; 
    RelManual_Out := FALSE;
    RelRemote_Out := FALSE;
	RelAuto_Out	  := FALSE;
	RelRemoteMobile_Out := FALSE; 
    HB_Manual_Out := FALSE;
	HB_Remote_Out := FALSE;
	HB_Auto_Out	  := FALSE;
	HB_Remote_Mobile_Out := FALSE; 
    RETURN;
END_IF

Valid         := TRUE;
ReqManual_Out := ReqManual;
ReqRemote_Out := ReqRemote;
ReqAuto_Out	  := ReqAuto;
ReqRemoteMobile_Out := ReqRemoteMobile;
AckManual_Out := AckManual;
AckRemote_Out := AckRemote;
AckAuto_Out	  := AckAuto;
AckRemoteMobile_Out := AckRemoteMobile; 
RelManual_Out := RelManual;
RelRemote_Out := RelRemote;
RelAuto_Out   := RelAuto;
RelRemoteMobile_Out := RelRemoteMobile; 
HB_Manual_Out := HB_Manual_Signal;
HB_Remote_Out := HB_Remote_Signal;
HB_Auto_Out	  := HB_Auto_Signal;
HB_Remote_Mobile_Out := HB_Remote_Mobile_Signal; 
                  
END_FUNCTION_BLOCK

FUNCTION_BLOCK DecisionLogger
  VAR_INPUT
    Active : EControlMode;
    Pending : EPendingMode;
    State : ETransitionState;
    RejectedRequestFlag : BOOL;
    RejectionReason : STRING;
  END_VAR
  VAR
    LastActive : EControlMode;
    LastPending : EPendingMode;
    LastState : ETransitionState;
    LastRejectedRequest : BOOL;
  END_VAR

                    IF Active <> LastActive THEN
		GVL_State.LastActiveBeforeTransition := LastActive;
END_IF
IF Active <> LastActive OR Pending <> LastPending OR State <> LastState THEN 
	GVL_State.Active := Active; 
	GVL_State.Pending := Pending; 
	GVL_State.State := State;

	LastActive := Active; 
 	LastPending := Pending; 
	LastState := State; 
END_IF

IF RejectedRequestFlag AND NOT LastRejectedRequest THEN
	GVL_State.RejectedRequestFlag := TRUE; //log the rejection
	GVL_State.RejectionReason := RejectionReason; 
END_IF
LastRejectedRequest := RejectedRequestFlag; 


                  
END_FUNCTION_BLOCK

CONFIGURATION CR710S
END_CONFIGURATION

CONFIGURATION SafetyPLC
  RESOURCE Application ON PLC
    {attribute 'location' := '16#800'}
    {attribute 'linkalways'}
    {attribute 'qualified_only'}
    VAR_GLOBAL  (* EVL - THIS EVL IS AUTOGENERATED. DO NOT MODIFY THESE ATTRIBUTES. *)
      HB_Manual_OK : BOOL;
      HB_Remote_OK : BOOL;
      HB_Auto_OK : BOOL;
      HB_Remote_Mobile_OK : BOOL;
    END_VAR
    TASK Task(INTERVAL := T#10ms, PRIORITY := 1);
    PROGRAM PLC_PRG WITH Task : PLC_PRG;
  END_RESOURCE
END_CONFIGURATION

CONFIGURATION Local_IO
END_CONFIGURATION

CONFIGURATION Inputs
END_CONFIGURATION

CONFIGURATION Outputs
END_CONFIGURATION

CONFIGURATION System_Inputs
END_CONFIGURATION

CONFIGURATION System_Outputs
END_CONFIGURATION

CONFIGURATION HMI
END_CONFIGURATION

CONFIGURATION User_LEDs
END_CONFIGURATION

CONFIGURATION Communication
END_CONFIGURATION

CONFIGURATION Ethernet
END_CONFIGURATION

CONFIGURATION CAN
END_CONFIGURATION

CONFIGURATION StandardPLC
  RESOURCE Application ON PLC
    {attribute 'qualified_only'}
    VAR_GLOBAL CONSTANT  (* GVL_HeartBeat *)
      HB_Generator_Interval : TIME := TIME#200ms;  (* HB_Generator_Interval must always be less than HB_Monitor_Timeout Current margin: 300ms - adjust both if either value changes *)
      HB_Monitor_Timeout : TIME := TIME#500ms;
      HB_Remote_Signal : BOOL;
      HB_Manual_Signal : BOOL;
      HB_Auto_Signal : BOOL;
      HB_Remote_Mobile_Signal : BOOL;
      HB_Manual_OK : BOOL;
      HB_Remote_OK : BOOL;
      HB_Auto_OK : BOOL;
      HB_Remote_Mobile_OK : BOOL;
    END_VAR
    {attribute 'qualified_only'}
    VAR_GLOBAL  (* GVL_IO *)
      ReqManual : BOOL;  (* Request *)
      ReqRemote : BOOL;
      ReqAuto : BOOL;
      ReqRemoteMobile : BOOL;
      AckManual : BOOL;  (* Acknowledge *)
      AckRemote : BOOL;
      AckAuto : BOOL;
      AckRemoteMobile : BOOL;
      RelManual : BOOL;  (* Release *)
      RelRemote : BOOL;
      RelAuto : BOOL;
      RelRemoteMobile : BOOL;
      ReleaseRequest_Manual : BOOL;
      ReleaseRequest_Remote : BOOL;
      Releaserequest_Auto : BOOL;
      ReleaseRequest_Remote_Mobile : BOOL;
    END_VAR
    {attribute 'qualified_only'}
    VAR_GLOBAL  (* GVL_State *)
      Active : EControlMode;  (* Currently active station *)
      Pending : EPendingMode;  (* Station wanting to take over *)
      State : ETransitionState;  (* Stable / Pending_Ack *)
      GrantedManual : BOOL;
      GrantedRemote : BOOL;
      GrantedAuto : BOOL;
      GrantedRemoteMobile : BOOL;
      Released : BOOL;
      PendingReady : BOOL;
      RejectedRequestFlag : BOOL;
      RejectionReason : STRING;
      LastActiveBeforeTransition : EControlMode;
      TimeStamp : UDINT;
    END_VAR
    TASK Task(INTERVAL := T#10ms, PRIORITY := 0);
    PROGRAM PLC_PRG WITH Task : PLC_PRG;
  END_RESOURCE
END_CONFIGURATION

CONFIGURATION Local_IO
END_CONFIGURATION

CONFIGURATION Inputs
END_CONFIGURATION

CONFIGURATION Outputs
END_CONFIGURATION

CONFIGURATION System_Inputs
END_CONFIGURATION

CONFIGURATION System_Outputs
END_CONFIGURATION

CONFIGURATION HMI
END_CONFIGURATION

CONFIGURATION User_LEDs
END_CONFIGURATION

CONFIGURATION Communication
END_CONFIGURATION

CONFIGURATION Ethernet
END_CONFIGURATION

CONFIGURATION CAN
END_CONFIGURATION
